PROGRAM V0_9
VAR
	fbRTrig : R_TRIG;
	bTrigger : BOOL;
	nState : SINT := 0;
END_VAR

(*
	Motor starten met één drukknop
	
	Schrijf een programma om een motor [ Relais voor MotorLinks en MotorRechts ] te starten en te stoppen met één drukknop. De installatie zal pas werken als een hoofdschakelaar AAN staat.
		1e druk op de drukknop:	start links draaiend
		2e druk op de drukknop:	stop
		3e druk op de drukknop:	start rechts draaiend
		4e druk op de drukknop:	stop
	
	bSwitch_1 = Hoofdschakelaar
	bButton_1 = Drukknop
	bLamp_1 = Links om
	bLamp_2 = Rechts om
*)

fbRTrig(CLK := GVL.bButton_1, Q => bTrigger);

END_PROGRAM

(* stored: Version 1.1.0.1, ProductVersion 3.1.4024.12
   POU V0_9: Id {57a44160-f458-495b-ab77-ebb92634c4d2}, SpecialFunc None *)
